Universal Robots PolyScope program: tb_retainer_and_nut_v2_hu.urp

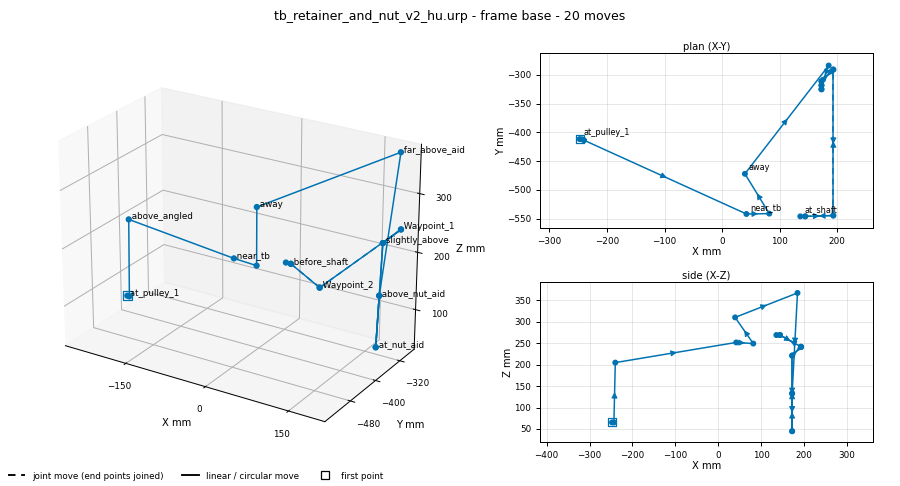
[picture p0: tool path of tb_retainer_and_nut_v2_hu.urp in frame base, 20 of 22 moves have a stored position in this frame; points joined in program order, loops and branches not executed]
Program tb_retainer_and_nut_v2_hu (installation=default directory=/programs/wrs2020 createdIn=5.6.0.90886 lastSavedIn=5.9.1.1031110 robotSerialNumber=20205500180)
Calibrated DH parameters: a=[0, -0.425, -0.3922, 0, 0, 0]; d=[0.1625, 0, 0, 0.1333, 0.0997, 0.0996]; alpha=[1.570796, 0, 0, 1.570796, -1.570796, 0]; deltaTheta=[0, 0, 0, 0, 0, 0]
Robot Program (runOnlyOnce=true)
  'Don't run. not complete'
  Halt
  current_pose := get_actual_tcp_pose()
  URCap Gripper (Robotiq_Grippers, Robotiq Inc.) dataModel(position=44.705882352941174, force=100.0, speed=100.0, positionInDouble=44.705882352941174, forceInDouble=100.0, speedInDouble=100.0, slaveIds=[9], blocking=true)
  MoveJ speed 60 deg/s, acceleration 80 deg/s^2 (useActiveTCP=true) feature=Base
    Waypoint at_pulley (Relative): relativeFromPosition TCP in base x=-247.499 y=-411.535 z=65.289 mm, rx=2.2244 ry=-2.2171 rz=-0.0362 rad; joints [43.772, -86.345, 117.338, -121.068, -91.318, -136.415] deg; TCP offset x=0 y=0 z=220 mm, rx=0 ry=0 rz=0 rad; TCP in base x=-247.495 y=-411.522 z=65.274 mm, rx=0.0051 ry=-3.1247 rz=-0.0246 rad; joints [43.771, -86.345, 117.34, -121.069, -91.317, -46.416] deg
  URCap Gripper (Robotiq_Grippers, Robotiq Inc.) dataModel(position=100.0, force=0.0, speed=0.0, positionInDouble=100.0, forceInDouble=0.0, speedInDouble=0.0, slaveIds=[9], blocking=true)
  URCap Gripper (Robotiq_Grippers, Robotiq Inc.) dataModel(position=45.09803921568627, force=0.0, speed=0.0, positionInDouble=45.09803921568627, forceInDouble=0.0, speedInDouble=0.0, slaveIds=[9], blocking=true)
  MoveJ speed 60 deg/s, acceleration 80 deg/s^2 (useActiveTCP=true) feature=Base
    Waypoint at_pulley (Relative): relativeFromPosition TCP in base x=-247.499 y=-411.535 z=65.289 mm, rx=2.2244 ry=-2.2171 rz=-0.0362 rad; joints [43.772, -86.345, 117.338, -121.068, -91.318, -136.415] deg; TCP in base x=-247.495 y=-411.522 z=65.274 mm, rx=0.0051 ry=-3.1247 rz=-0.0246 rad; joints [43.771, -86.345, 117.34, -121.069, -91.317, -46.416] deg
  SuppressedNode
    MoveJ speed 180 deg/s, acceleration 150 deg/s^2 (useActiveTCP=false) tcp=gripper_140_tip; feature=Base
      Waypoint home: TCP in base x=133.727 y=-178.735 z=460.339 mm, rx=-0.0013 ry=3.138 rz=0.0408 rad; joints [90.031, -120.136, 80.128, -48.416, -89.757, -0.16] deg; TCP offset x=0 y=0 z=220 mm, rx=0 ry=0 rz=0 rad
  SuppressedNode
    MoveJ speed 180 deg/s, acceleration 150 deg/s^2 (useActiveTCP=true) feature=Base
      Waypoint Waypoint_12: TCP in base x=-82.102 y=-275.549 z=387.348 mm, rx=-0.1814 ry=-3.1114 rz=0.2863 rad; joints [35.849, -127.007, 98.51, -68.6, -82.206, -47.132] deg; TCP offset x=0 y=0 z=220 mm, rx=0 ry=0 rz=0 rad
  SuppressedNode
    MoveJ speed 180 deg/s, acceleration 150 deg/s^2 (useActiveTCP=true) feature=Base
      Waypoint above_idler: TCP in base x=-247.479 y=-411.551 z=212.636 mm, rx=2.2243 ry=-2.2171 rz=-0.0361 rad; joints [43.828, -93.41, 101.402, -97.983, -91.147, -136.367] deg
  SuppressedNode
    MoveL speed 50 mm/s, acceleration 1200 mm/s^2 (useActiveTCP=true) feature=Base
      Waypoint at_pulley_1: motionParameters(jointSpeed=1.047198 jointAcceleration=1.396263 cartesianSpeed=0.5 cartesianAcceleration=1.2); TCP in base x=-247.479 y=-411.551 z=65.293 mm, rx=2.2243 ry=-2.2171 rz=-0.0361 rad; joints [43.809, -86.378, 117.317, -120.929, -91.133, -136.311] deg
  SuppressedNode
    MoveL speed 50 mm/s, acceleration 1200 mm/s^2 (useActiveTCP=true) feature=Base
      Waypoint Waypoint (Variable): motionParameters(jointSpeed=1.047198 jointAcceleration=1.396263 cartesianSpeed=0.5 cartesianAcceleration=1.2)
  URCap Gripper (Robotiq_Grippers, Robotiq Inc.) dataModel(position=100.0, force=0.0, speed=0.0, positionInDouble=100.0, forceInDouble=0.0, speedInDouble=0.0, slaveIds=[9], blocking=true)
  URCap Gripper (Robotiq_Grippers, Robotiq Inc.) dataModel(position=57.64705882352941, force=0.0, speed=0.0, positionInDouble=57.64705882352941, forceInDouble=0.0, speedInDouble=0.0, slaveIds=[9], blocking=true)
  MoveL speed 50 mm/s, acceleration 1200 mm/s^2 (useActiveTCP=true) feature=Base
    Waypoint at_pulley_1: motionParameters(jointSpeed=1.047198 jointAcceleration=1.396263 cartesianSpeed=0.5 cartesianAcceleration=1.2); TCP in base x=-247.479 y=-411.551 z=65.293 mm, rx=2.2243 ry=-2.2171 rz=-0.0361 rad; joints [43.809, -86.378, 117.317, -120.929, -91.133, -136.311] deg
  MoveL speed 50 mm/s, acceleration 1200 mm/s^2 (useActiveTCP=true) feature=Base
    Waypoint angled: motionParameters(jointSpeed=1.047198 jointAcceleration=1.396263 cartesianSpeed=0.5 cartesianAcceleration=1.2); TCP in base x=-243.13 y=-411.958 z=65.291 mm, rx=1.8379 ry=-1.8459 rz=-0.6644 rad; joints [65.515, -83.312, 132.748, -156.267, -125.111, -119.597] deg; TCP offset x=0 y=0 z=220 mm, rx=0 ry=0 rz=0 rad
  URCap Gripper (Robotiq_Grippers, Robotiq Inc.) dataModel(position=100.0, force=0.0, speed=0.0, positionInDouble=100.0, forceInDouble=0.0, speedInDouble=0.0, slaveIds=[9], blocking=true)
  MoveL speed 250 mm/s, acceleration 1200 mm/s^2 (useActiveTCP=true) feature=Base
    Waypoint above_angled: motionParameters(jointSpeed=1.047198 jointAcceleration=1.396263 cartesianSpeed=0.25 cartesianAcceleration=1.2); TCP in base x=-239.887 y=-413.598 z=204.833 mm, rx=1.8379 ry=-1.8459 rz=-0.6644 rad; joints [66.077, -97.285, 120.862, -129.87, -125.089, -118.783] deg; TCP offset x=0 y=0 z=220 mm, rx=0 ry=0 rz=0 rad
    Waypoint near_tb: motionParameters(blendRadius=0.038); TCP in base x=42.161 y=-541.658 z=251.88 mm, rx=-2.2078 ry=1.5258 rz=-1.5075 rad; joints [47.035, -95.124, 115.286, -91.003, -33.11, -164.164] deg
    Waypoint in_ridge: motionParameters(jointSpeed=1.047198 jointAcceleration=1.396263 cartesianSpeed=0.02 cartesianAcceleration=1.2); TCP in base x=81.893 y=-541.004 z=249.227 mm, rx=-2.2078 ry=1.5258 rz=-1.5075 rad; joints [51.109, -97.259, 119.171, -98.883, -31.982, -156.881] deg
  Popup Message (haltProgram=false message=wait for screw tool to hold inputType=Text)
  URCap Gripper (Robotiq_Grippers, Robotiq Inc.) dataModel(position=41.96078431372549, force=100.0, speed=100.0, positionInDouble=41.96078431372549, forceInDouble=100.0, speedInDouble=100.0, slaveIds=[9], blocking=true)
  MoveL speed 250 mm/s, acceleration 1200 mm/s^2 (useActiveTCP=true) feature=Base
    Waypoint away: TCP in base x=39.547 y=-471.894 z=310.294 mm, rx=-2.2141 ry=1.5067 rz=-1.5032 rad; joints [39.591, -105.138, 111.963, -66.814, -36.61, -177.398] deg
    Waypoint far_above_aid: TCP in base x=185.019 y=-283.793 z=367.304 mm, rx=3.0427 ry=0.0266 rz=0.0843 rad; joints [97.518, -117.381, 97.301, -75.775, -87.414, -173.456] deg
  MoveL speed 250 mm/s, acceleration 1200 mm/s^2 (useActiveTCP=true) feature=Base
    Waypoint above_nut_aid: TCP in base x=172.519 y=-318.273 z=132.878 mm, rx=3.1334 ry=-0.0123 rz=-0.0179 rad; joints [97.626, -109.17, 125.745, -106.863, -90.541, -171.937] deg
    URCap Gripper (Robotiq_Grippers, Robotiq Inc.) dataModel(position=21.96078431372549, force=100.0, speed=100.0, positionInDouble=21.96078431372549, forceInDouble=100.0, speedInDouble=100.0, slaveIds=[9], blocking=true)
    Waypoint at_nut_aid: TCP in base x=172.519 y=-325.105 z=44.86 mm, rx=3.1334 ry=-0.0123 rz=-0.0179 rad; joints [97.451, -101.585, 134.781, -123.486, -90.53, -172.054] deg
    URCap Gripper (Robotiq_Grippers, Robotiq Inc.) dataModel(position=100.0, force=100.0, speed=100.0, positionInDouble=100.0, forceInDouble=100.0, speedInDouble=100.0, slaveIds=[9], blocking=true)
    Waypoint slightly_above: TCP in base x=172.519 y=-311.073 z=221.087 mm, rx=3.1334 ry=-0.0123 rz=-0.0179 rad; joints [97.806, -112.461, 114.667, -92.492, -90.559, -171.799] deg
  MoveL speed 250 mm/s, acceleration 1200 mm/s^2 (useActiveTCP=true) feature=Base
    Waypoint Waypoint_1: TCP in base x=193.098 y=-290.824 z=241.653 mm, rx=-2.26 ry=-2.0992 rz=0.0999 rad; joints [105.872, -111.142, 110.658, -88.291, -94.599, -249.911] deg
    Waypoint Waypoint_2: motionParameters(blendRadius=0.036); TCP in base x=193.098 y=-544.308 z=241.653 mm, rx=-2.26 ry=-2.0992 rz=0.0999 rad; joints [98.952, -79.277, 82.032, -92.106, -94.688, -256.794] deg
    Waypoint before_shaft: TCP in base x=144.255 y=-545.79 z=269.11 mm, rx=2.2425 ry=2.1895 rz=-0.0818 rad; joints [92.327, -83.742, 83.817, -92.266, -91.814, -266.35] deg; TCP offset x=0 y=0 z=220 mm, rx=0 ry=0 rz=0 rad
  MoveL speed 5 mm/s, acceleration 100 mm/s^2 (useActiveTCP=true) feature=Base
    Waypoint at_shaft: TCP in base x=135.746 y=-545.79 z=269.11 mm, rx=2.2425 ry=2.1895 rz=-0.0818 rad; joints [91.42, -84.064, 84.185, -92.342, -91.778, -267.256] deg; TCP offset x=0 y=0 z=220 mm, rx=0 ry=0 rz=0 rad
    Popup Message (haltProgram=false message=turn on motor, then press enter to start spiral motion inputType=Text)
    Force Frame feature=Base; selection=[1, 0, 0, 0, 0, 0]; wrench=[-5, 0, 10, 0, 0, 0]; limitsForce=[0.005, 0.15, 0.01, 1.047198, 1.047198, 1.047198]; limitsMotion=[0.1, 0.1, 0.1, 0.349066, 0.349066, 0.349066]
      Loop Counting (count=5) loopVariable(name=Loop_1)
        MoveDirectionNode (selectedDirection=YPlus) feature=Base
          Until DISTANCE (allowActions=false deceleration=3 distanceNodeType=STOP) Distance=0.002; motionParameters(blendRadius=0)
        MoveDirectionNode (selectedDirection=ZPlus) feature=Base
          Until DISTANCE (allowActions=false deceleration=3 distanceNodeType=STOP) Distance=0.002; motionParameters(blendRadius=0)
        MoveDirectionNode (selectedDirection=YMinus) feature=Base
          Until DISTANCE (allowActions=false deceleration=3 distanceNodeType=STOP) Distance=0.002; motionParameters(blendRadius=0)
        MoveDirectionNode (selectedDirection=YMinus) feature=Base
          Until DISTANCE (allowActions=false deceleration=3 distanceNodeType=STOP) Distance=0.002; motionParameters(blendRadius=0)
        MoveDirectionNode (selectedDirection=ZMinus) feature=Base
          Until DISTANCE (allowActions=false deceleration=3 distanceNodeType=STOP) Distance=0.002; motionParameters(blendRadius=0)
        MoveDirectionNode (selectedDirection=YPlus) feature=Base
          Until DISTANCE (allowActions=false deceleration=3 distanceNodeType=STOP) Distance=0.002; motionParameters(blendRadius=0)
        MoveDirectionNode (selectedDirection=YPlus) feature=Base
          Until DISTANCE (allowActions=false deceleration=3 distanceNodeType=STOP) Distance=0.002; motionParameters(blendRadius=0)
        MoveDirectionNode (selectedDirection=ZMinus) feature=Base
          Until DISTANCE (allowActions=false deceleration=3 distanceNodeType=STOP) Distance=0.002; motionParameters(blendRadius=0)
        MoveDirectionNode (selectedDirection=YMinus) feature=Base
          Until DISTANCE (allowActions=false deceleration=3 distanceNodeType=STOP) Distance=0.002; motionParameters(blendRadius=0)
        MoveDirectionNode (selectedDirection=YMinus) feature=Base
          Until DISTANCE (allowActions=false deceleration=3 distanceNodeType=STOP) Distance=0.002; motionParameters(blendRadius=0)
        MoveDirectionNode (selectedDirection=ZPlus) feature=Base
          Until DISTANCE (allowActions=false deceleration=3 distanceNodeType=STOP) Distance=0.002; motionParameters(blendRadius=0)
        MoveDirectionNode (selectedDirection=YPlus) feature=Base
          Until DISTANCE (allowActions=false deceleration=3 distanceNodeType=STOP) Distance=0.002; motionParameters(blendRadius=0)
  Popup Message (haltProgram=false message=ok? inputType=Text)
  MoveJ speed 60 deg/s, acceleration 80 deg/s^2 (useActiveTCP=true) feature=Base
    Waypoint before_shaft: motionParameters(jointSpeed=1.047198 jointAcceleration=1.396263 cartesianSpeed=0.25 cartesianAcceleration=1.2); TCP in base x=144.255 y=-545.79 z=269.11 mm, rx=2.2425 ry=2.1895 rz=-0.0818 rad; joints [92.327, -83.742, 83.817, -92.266, -91.814, -266.35] deg; TCP offset x=0 y=0 z=220 mm, rx=0 ry=0 rz=0 rad
    Waypoint Waypoint_2: motionParameters(jointSpeed=2.094395 jointAcceleration=2.094395 cartesianSpeed=0.25 cartesianAcceleration=1.2 blendRadius=0.05); TCP in base x=193.098 y=-544.308 z=241.653 mm, rx=-2.26 ry=-2.0992 rz=0.0999 rad; joints [98.952, -79.277, 82.032, -92.106, -94.688, -256.794] deg; TCP offset x=0 y=0 z=220 mm, rx=0 ry=0 rz=0 rad
    Waypoint Waypoint_1: motionParameters(jointSpeed=2.094395 jointAcceleration=2.094395 cartesianSpeed=0.25 cartesianAcceleration=1.2); TCP in base x=193.098 y=-290.824 z=241.653 mm, rx=-2.26 ry=-2.0992 rz=0.0999 rad; joints [105.872, -111.142, 110.658, -88.291, -94.599, -249.911] deg
  MoveL speed 250 mm/s, acceleration 1200 mm/s^2 (useActiveTCP=true) feature=Base
    Waypoint slightly_above: TCP in base x=172.519 y=-311.073 z=221.087 mm, rx=3.1334 ry=-0.0123 rz=-0.0179 rad; joints [97.806, -112.461, 114.667, -92.492, -90.559, -171.799] deg
    Waypoint at_nut_aid: TCP in base x=172.519 y=-325.105 z=44.86 mm, rx=3.1334 ry=-0.0123 rz=-0.0179 rad; joints [97.451, -101.585, 134.781, -123.486, -90.53, -172.054] deg
    URCap Gripper (Robotiq_Grippers, Robotiq Inc.) dataModel(position=21.96078431372549, force=100.0, speed=100.0, positionInDouble=21.96078431372549, forceInDouble=100.0, speedInDouble=100.0, slaveIds=[9], blocking=true)
    Waypoint above_nut_aid: TCP in base x=172.519 y=-318.273 z=132.878 mm, rx=3.1334 ry=-0.0123 rz=-0.0179 rad; joints [97.626, -109.17, 125.745, -106.863, -90.541, -171.937] deg
